(* PLC project Tc2_Utilities.FB_StringRingBuffer Demo, tc3-libraries-kb TwinCAT 3.1 *)
(* stored: creationDateTime 2026-05-10T20:00:00, modificationDateTime 2026-05-10T20:00:00 *)

PROGRAM P_Demo_FB_StringRingBuffer
  VAR
    fbFB_StringRingBuffer : FB_StringRingBuffer;  (* Tc2_Utilities.FB_StringRingBuffer 实例 *)
    arg_bOverwrite : BOOL;  (* VAR_INPUT bOverwrite *)
    arg_putValue : T_MaxString;  (* VAR_INPUT putValue *)
    arg_pBuffer : POINTER TO BYTE;  (* VAR_INPUT pBuffer *)
    arg_cbBuffer : UDINT;  (* VAR_INPUT cbBuffer *)
    out_bOk : BOOL;  (* VAR_OUTPUT bOk *)
    out_getValue : T_MaxString;  (* VAR_OUTPUT getValue *)
    out_nCount : UDINT;  (* VAR_OUTPUT nCount *)
    out_cbSize : UDINT;  (* VAR_OUTPUT cbSize *)
  END_VAR

            // ============================================================
// Tc2_Utilities.FB_StringRingBuffer 演示程序（FB 实例）
// ============================================================
// 验证步骤：
//   1. 引用 Tc2_Utilities（及依赖类型所在库 Tc2_System 等）
//   2. 编译 + 登录
//   3. 按 doc.md 给 arg_* 赋值
//   4. 在线监视 out_* / io_* 输出
// ============================================================

fbFB_StringRingBuffer(
    bOverwrite := arg_bOverwrite,
    putValue := arg_putValue,
    pBuffer := arg_pBuffer,
    cbBuffer := arg_cbBuffer,
    bOk => out_bOk,
    getValue => out_getValue,
    nCount => out_nCount,
    cbSize => out_cbSize
);

          
END_PROGRAM
